// Block: RollformerLubr_PERS

DATA_BLOCK RollformerLubr_PERS
VERSION : 0.1
   NON_RETAIN
   VAR
      Pump : LubrMotor_Par;
      Valves1 : Struct
         Control : LubrValve_Pers;
         Enable_V : Array[1..ROLL_LUBR_MAXVALVE] of Bool;
      END_STRUCT;
      Valves2 : Struct
         Control : LubrValve_Pers;
         Enable_V : Array[1..ROLL_LUBR_MAXVALVE] of Bool;
      END_STRUCT;
      Valves3 : Struct
         Control : LubrValve_Pers;
         Enable_V : Array[1..ROLL_LUBR_MAXVALVE] of Bool;
      END_STRUCT;
   END_VAR

BEGIN
   // No initialization required
END_DATA_BLOCK
